% RSLogix 500 project PUMPVALVE.RSS, saved by version 8.30.00.16 %
PROJECT "UNTITLED"    % processor: Bul.1763 MicroLogix 1100 Series B %

PROGRAM FILES
  LAD 2 "MAIN"  4 rungs
  LAD 3 "I/O"  7 rungs
  LAD 4 "ALARMS"  7 rungs
  LAD 5 "CONTROLS"  5 rungs

DATA FILES
  O0 OUTPUT  5 elements
  I1 INPUT  7 elements
  S2 STATUS  66 elements
  B3 BINARY  2 elements
  T4 TIMER  4 elements
  C5 COUNTER  1 elements
  R6 CONTROL  1 elements
  N7 INTEGER  1 elements
  F8 FLOAT  1 elements

LADDER 2 "MAIN"
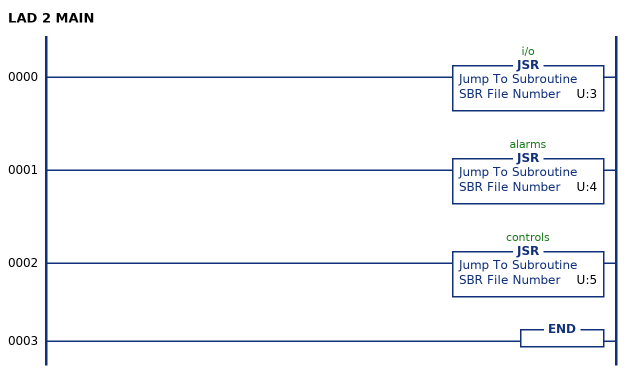
% Rung: 0 %
SOR JSR U:3 EOR
%   U:3  "i/o" %
% Rung: 1 %
SOR JSR U:4 EOR
%   U:4  "alarms" %
% Rung: 2 %
SOR JSR U:5 EOR
%   U:5  "controls" %
% Rung: 3 %
SOR END EOR

LADDER 3 "I/O"
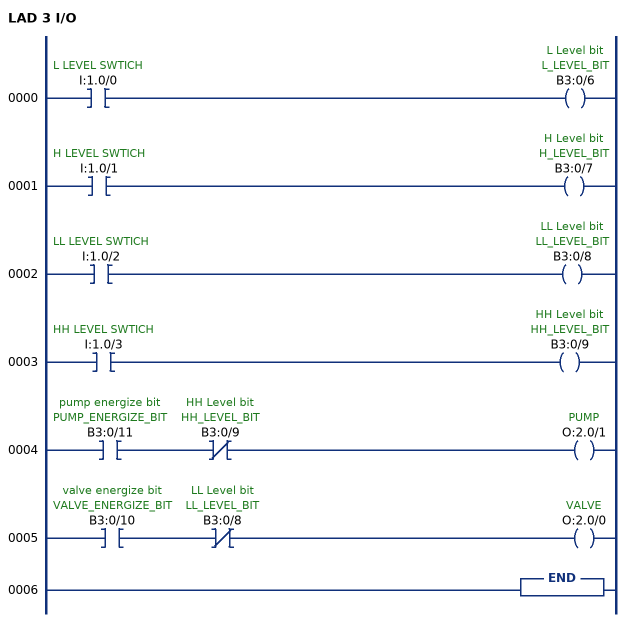
% Rung: 0 %
SOR XIC I:1.0/0 OTE B3:0/6 EOR
%   I:1.0/0  "L LEVEL SWTICH" %
%   B3:0/6  L_LEVEL_BIT  "L Level bit" %
% Rung: 1 %
SOR XIC I:1.0/1 OTE B3:0/7 EOR
%   I:1.0/1  "H LEVEL SWTICH" %
%   B3:0/7  H_LEVEL_BIT  "H Level bit" %
% Rung: 2 %
SOR XIC I:1.0/2 OTE B3:0/8 EOR
%   I:1.0/2  "LL LEVEL SWTICH" %
%   B3:0/8  LL_LEVEL_BIT  "LL Level bit" %
% Rung: 3 %
SOR XIC I:1.0/3 OTE B3:0/9 EOR
%   I:1.0/3  "HH LEVEL SWTICH" %
%   B3:0/9  HH_LEVEL_BIT  "HH Level bit" %
% Rung: 4 %
SOR XIC B3:0/11 XIO B3:0/9 OTE O:2.0/1 EOR
%   B3:0/11  PUMP_ENERGIZE_BIT  "pump energize bit" %
%   B3:0/9  HH_LEVEL_BIT  "HH Level bit" %
%   O:2.0/1  "PUMP" %
% Rung: 5 %
SOR XIC B3:0/10 XIO B3:0/8 OTE O:2.0/0 EOR
%   B3:0/10  VALVE_ENERGIZE_BIT  "valve energize bit" %
%   B3:0/8  LL_LEVEL_BIT  "LL Level bit" %
%   O:2.0/0  "VALVE" %
% Rung: 6 %
SOR END EOR

LADDER 4 "ALARMS"
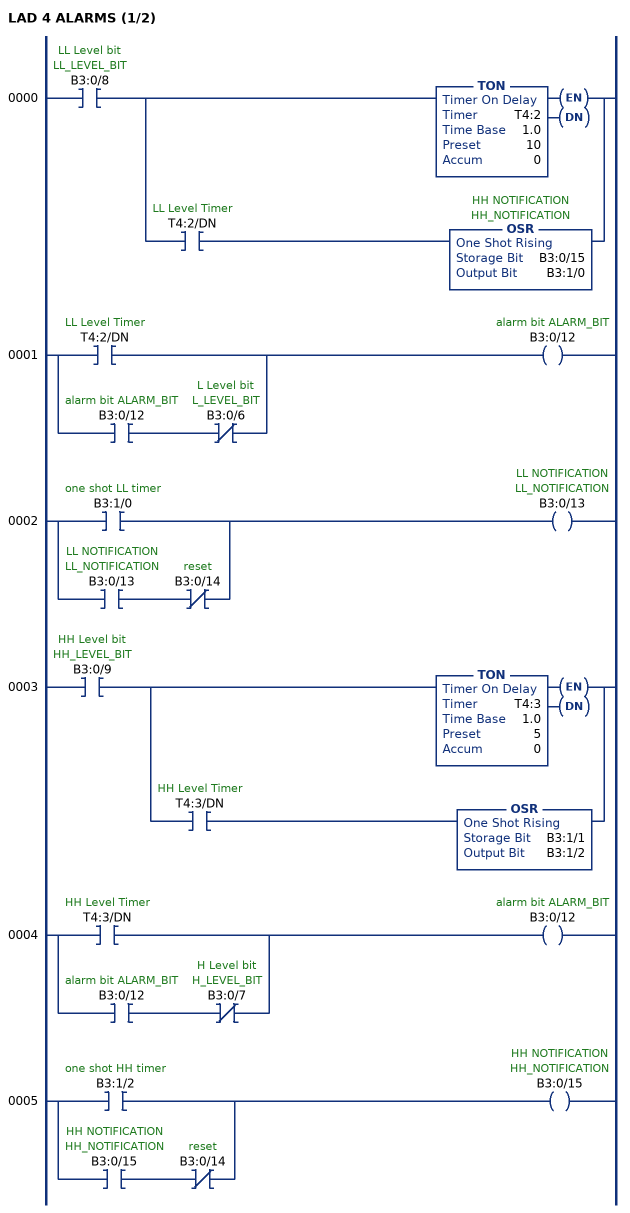
% Rung: 0 %
SOR XIC B3:0/8 BST TON T4:2 1.0 10 0 NXB XIC T4:2/DN OSR B3:0/15 B3:1/0 BND EOR
%   B3:0/8  LL_LEVEL_BIT  "LL Level bit" %
%   T4:2/DN  "LL Level Timer" %
%   B3:0/15  HH_NOTIFICATION  "HH NOTIFICATION" %
%   B3:1/0  "one shot LL timer" %
% Rung: 1 %
SOR BST XIC T4:2/DN NXB XIC B3:0/12 XIO B3:0/6 BND OTE B3:0/12 EOR
%   T4:2/DN  "LL Level Timer" %
%   B3:0/12  ALARM_BIT  "alarm bit" %
%   B3:0/6  L_LEVEL_BIT  "L Level bit" %
% Rung: 2 %
SOR BST XIC B3:1/0 NXB XIC B3:0/13 XIO B3:0/14 BND OTE B3:0/13 EOR
%   B3:1/0  "one shot LL timer" %
%   B3:0/13  LL_NOTIFICATION  "LL NOTIFICATION" %
%   B3:0/14  "reset" %
% Rung: 3 %
SOR XIC B3:0/9 BST TON T4:3 1.0 5 0 NXB XIC T4:3/DN OSR B3:1/1 B3:1/2 BND EOR
%   B3:0/9  HH_LEVEL_BIT  "HH Level bit" %
%   T4:3/DN  "HH Level Timer" %
%   B3:1/2  "one shot HH timer" %
% Rung: 4 %
SOR BST XIC T4:3/DN NXB XIC B3:0/12 XIO B3:0/7 BND OTE B3:0/12 EOR
%   T4:3/DN  "HH Level Timer" %
%   B3:0/12  ALARM_BIT  "alarm bit" %
%   B3:0/7  H_LEVEL_BIT  "H Level bit" %
% Rung: 5 %
SOR BST XIC B3:1/2 NXB XIC B3:0/15 XIO B3:0/14 BND OTE B3:0/15 EOR
%   B3:1/2  "one shot HH timer" %
%   B3:0/15  HH_NOTIFICATION  "HH NOTIFICATION" %
%   B3:0/14  "reset" %

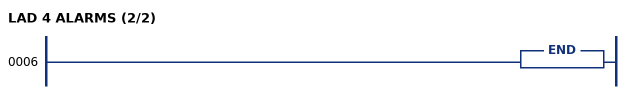
% Rung: 6 %
SOR END EOR

LADDER 5 "CONTROLS"
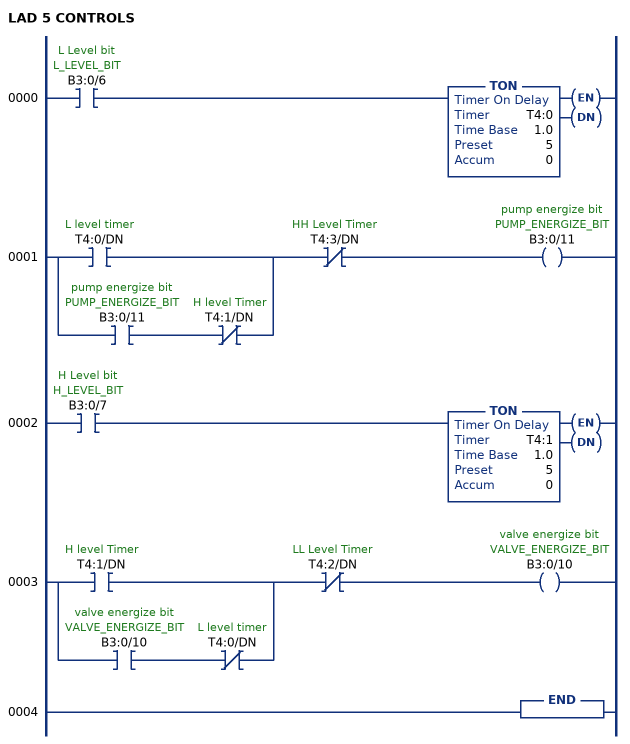
% Rung: 0 %
SOR XIC B3:0/6 TON T4:0 1.0 5 0 EOR
%   B3:0/6  L_LEVEL_BIT  "L Level bit" %
% Rung: 1 %
SOR BST XIC T4:0/DN NXB XIC B3:0/11 XIO T4:1/DN BND XIO T4:3/DN OTE B3:0/11 EOR
%   T4:0/DN  "L level timer" %
%   B3:0/11  PUMP_ENERGIZE_BIT  "pump energize bit" %
%   T4:1/DN  "H level Timer" %
%   T4:3/DN  "HH Level Timer" %
% Rung: 2 %
SOR XIC B3:0/7 TON T4:1 1.0 5 0 EOR
%   B3:0/7  H_LEVEL_BIT  "H Level bit" %
% Rung: 3 %
SOR BST XIC T4:1/DN NXB XIC B3:0/10 XIO T4:0/DN BND XIO T4:2/DN OTE B3:0/10 EOR
%   T4:1/DN  "H level Timer" %
%   B3:0/10  VALVE_ENERGIZE_BIT  "valve energize bit" %
%   T4:0/DN  "L level timer" %
%   T4:2/DN  "LL Level Timer" %
% Rung: 4 %
SOR END EOR

OTHER DOCUMENTED ADDRESSES
  B3:0/0  "L Level"
  B3:0/1  "H Level"
  B3:0/2  "LL Level"
  B3:0/3  "HH Level"
  B3:0/4  "valve"
  B3:0/5  "pump"
  B3:1/3  "LL ons bit"
  B3:1/4  "hh ons bit"
  B3:1/6  "hh osr bit"
  B3:1/7  "ll osr bit"
  I:0.0/0  "L level switch"
  I:0.0/1  "H level switch"
  I:0.0/2  "LL level switch"
  I:0.0/3  "HH level switch"
  O:0.0/0  "valve"
  O:0.0/1  "pump"

DATA TABLE (non-zero values as saved)
DATA T4
% .PRE .ACC %
% T4:0 % 5 0
% T4:1 % 5 0
% T4:2 % 10 0
% T4:3 % 5 0
